(* IEC 61131-3 sources: RL_MAR/experiments/comparison/llm4plc/results/deepseek-ai-DeepSeek-V3.2_20260506_104945/20260506_121930, 1 file *)

(* ---- generated_code_iteration_0.st ---- *)
START_ST
FUNCTION_BLOCK FB_ConditionalSelectAndAggregate
VAR_INPUT
Z : INT;
END_VAR
VAR
A_X : INT := 42;
A_Y : INT := 333;
tempSelected : INT;
END_VAR
VAR_OUTPUT
NEW_Z : INT;
END_VAR

IF A_X > Z THEN
    tempSelected := A_Y;
ELSE
    tempSelected := Z;
END_IF;
NEW_Z := tempSelected + A_X + A_Y;

END_FUNCTION_BLOCK
END_ST
